PROGRAM MAIN
VAR
	nFactorial : ULINT;
	Profiler : PROFILER;
	ProfilerResult : PROFILERSTRUCT;
END_VAR

Profiler(START := TRUE, RESET := FALSE);
Factorial(n := nFactorial);
Profiler(START := FALSE);
ProfilerResult := Profiler.DATA;

END_PROGRAM

(* stored: Version 1.1.0.1, ProductVersion 3.1.4024.12
   POU MAIN: Id {bbfefc72-33fb-4904-9bd7-b243dcfdea99}, SpecialFunc None *)
